// TwinCAT 3 PLC project xae_ads_client_test_plc
// ProgramVersion: 3.1.4024.0
// libraries:
//   Tc2_Standard, * (Beckhoff Automation GmbH)
//   Tc2_System, * (Beckhoff Automation GmbH)
//   Tc3_Module, * (Beckhoff Automation GmbH)
// project tree:
//   DUTs/ E_TestEnum.TcDUT, ST_Example.TcDUT
//   GVLs/ GVL_Test.TcGVL
//   / PlcTask.TcTTO
//   POUs/ MAIN.TcPOU
// real-time tasks:
//   TASK PlcTask: cycle T#10ms, priority 20, ADS port 350

CONFIGURATION xae_ads_client_test_plc
    RESOURCE PLC ON TwinCAT3
        TASK PlcTask(INTERVAL := T#10ms, PRIORITY := 20);
        PROGRAM MAIN WITH PlcTask : MAIN;
    END_RESOURCE
END_CONFIGURATION

// ---- DUTs/E_TestEnum.TcDUT
{attribute 'qualified_only'}
{attribute 'strict'}
TYPE E_TestEnum :
(
	Disabled 	:= 0,
	Starting 	:= 50,
	Running 	:= 100,
	Stopping	:= 200	
);
END_TYPE

// ---- DUTs/ST_Example.TcDUT
TYPE ST_Example :
STRUCT
	SomeText : STRING(50) := 'Hello ads-client';
	SomeReal : REAL := 3.14159265359;
	SomeDate : DT := DT#2020-4-13-12:25:33;
END_STRUCT
END_TYPE

// ---- GVLs/GVL_Test.TcGVL
{attribute 'qualified_only'}
//GVL_Test
VAR_GLOBAL
  TestINT           : INT := 1234;
  TestSTRING        : STRING := 'Hello this is a test string';
  ExampleSTRUCT     : ST_Example;
  TestARRAY         : ARRAY[0..4] OF INT := [0, 10, 200, 3000, 4000];
  TestARRAY2        : ARRAY[0..4] OF ST_Example := [(SomeText := 'Just for demo purposes')];
  TestENUM          : E_TestEnum := E_TestEnum.Running;
  IncrementingValue : INT; //This should change every 500 ms or so
  TestTimer         : TON := (PT := T#2S500MS);
END_VAR

// ---- POUs/MAIN.TcPOU
PROGRAM MAIN
VAR
	cnt : DINT;
END_VAR

cnt := cnt + 1;

END_PROGRAM
